(* PLC project Unnamed, Unknown Unnamed 1 *)
(* stored: creationDateTime 2025-11-04T16:29:39, modificationDateTime 2025-11-04T16:34:44 *)

PROGRAM main
  VAR NON_RETAIN
    Trigger : BOOL := False;
    SealedInCoil : BOOL := False;
  END_VAR

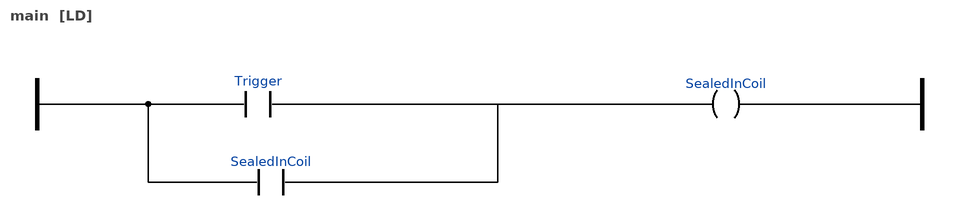
(* LD diagram, written out as Structured Text *)
SealedInCoil := Trigger OR SealedInCoil;
END_PROGRAM

CONFIGURATION Config0
  RESOURCE Res0 ON PLC
    TASK task0(INTERVAL := T#20ms, PRIORITY := 0);
    PROGRAM instance0 : main;
  END_RESOURCE
END_CONFIGURATION
